// TIA Portal V20 export
TYPE "LER_typeSleepModeParameter"
// stored: Access Published
   STRUCT
      sleepMode : Struct
         "time" : Time;
         ffu : Int;
         ringBlower : Real;
         heater : Int;
      END_STRUCT;
      DeepsleepMode : Struct
         "time" : Time;
         ffu : Int;
         ringBlower : Real;
         heater : Int;
      END_STRUCT;
   END_STRUCT;
END_TYPE
